// Mitsubishi GX Works2 project: v05   PLC: Q02/Q02H

PROGRAM MAIN
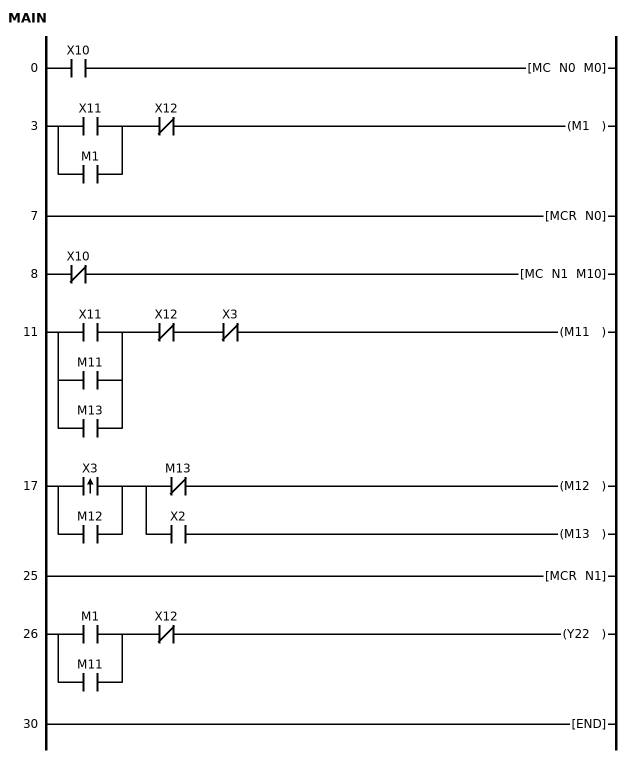
0     LD      X10
      MC      N0 M0
3     LD      X11
      OR      M1
      ANI     X12
      OUT     M1
7     MCR     N0
8     LDI     X10
      MC      N1 M10
11    LD      X11
      OR      M11
      OR      M13
      ANI     X12
      ANI     X3
      OUT     M11
17    LDP     X3
      OR      M12
      MPS
      ANI     M13
      OUT     M12
      MPP
      AND     X2
      OUT     M13
25    MCR     N1
26    LD      M1
      OR      M11
      ANI     X12
      OUT     Y22
30    END
END_PROGRAM
